FUNCTION_BLOCK FB_EcoWash IMPLEMENTS I_WashStrategy
VAR
	stWashSettings : ST_WashSettings;
END_VAR

METHOD FB_init : BOOL
VAR_INPUT
	bInitRetains : BOOL; // if TRUE, the retain variables are initialized (warm start / cold start)
	bInCopyCode : BOOL;  // if TRUE, the instance afterwards gets moved into the copy code (online change)
END_VAR
IF stWashSettings.sDescription = '' THEN
	stWashSettings.rWashTemperature := GVL_WashConstants.ECO_TEMP;
	stWashSettings.nSpinSpeed:= GVL_WashConstants.ECO_SPIN;
	stWashSettings.tWashDuration := GVL_WashConstants.ECO_WASH_TIME;
	stWashSettings.sDescription := GVL_WashConstants.ECO_DESC;
	
END_IF

FB_init :=TRUE;
END_METHOD

{warning 'add method implementation '}
METHOD GetProgramName : STRING
GetProgramName := 'Eco';
END_METHOD

METHOD GetRinseTime : TIME
VAR_INPUT
END_VAR
GetRinseTime := GVL_WashConstants.ECO_WASH_RINSE_TIME;
END_METHOD

METHOD GetSpinTime :  TIME
VAR_INPUT
	
END_VAR
GetSpinTime := GVL_WashConstants.ECO_WASH_SPIN_TIME;
END_METHOD


METHOD GetWashSettings :  ST_WashSettings
GetWashSettings := stWashSettings;
END_METHOD

END_FUNCTION_BLOCK

(* stored: Version 1.1.0.1, ProductVersion 3.1.4024.16
   POU FB_EcoWash: Id {1835ade7-aea4-4535-b27c-cd26b020b72e}, SpecialFunc None
   Method FB_init: Id {c98c696c-81fe-4c7a-9ec2-39f1f1acbc87}
   Method GetProgramName: Id {ec403252-a071-4ef3-8743-81c62b8e8044}
   Method GetRinseTime: Id {716d5d1b-d1b6-4b13-bb20-a4bfd680c553}
   Method GetSpinTime: Id {e5f5115f-2297-4a11-84f8-ca9301a51234}
   Method GetWashSettings: Id {6b162565-bd4d-43c4-912d-4109d36d718a} *)
